// TIA Portal V15.1 export
// export: Created 2026-01-09T13:45:15.6924077Z, ExportSetting WithDefaults, WithReadOnly, DisplayName Totally Integrated Automation Portal, DisplayVersion V15.1 Update 8, DisplayName TIA Portal Openness, DisplayVersion V15.1 Update 8, DisplayName STEP 7 Professional, DisplayVersion V15.1 Update 8, DisplayName WinCC Advanced, DisplayVersion V15.1 Update 8
FUNCTION "FCXL_CCD_AP1" : Void   // FC15, LAD
{ S7_Optimized_Access := 'TRUE' }
VERSION : 0.1
// stored: AutoNumber true, CodeModifiedDate 2026-01-04T14:27:05.6438339Z, CompileDate 2026-01-04T14:27:05.690726Z, CreationDate 2024-10-13T15:07:34.9617085Z, HandleErrorsWithinBlock false, InterfaceModifiedDate 2024-08-08T03:23:40.7447783Z, IsConsistent true, IsIECCheckEnabled false, IsKnowHowProtected false, IsWriteProtected false, LibraryConformanceStatus Error: The block contains calls of single instances. Warning: The object contains access to global data blocks. Warning: The block contains direct access to inputs, outputs, bit memories, indirect access to the registry or indirect access to external memory areas that are unknown at the time of compilation., ModifiedDate 2026-01-04T14:27:05.6438339Z, ParameterModified 2024-08-08T03:23:40.7447783Z, PLCSimAdvancedSupport false, SetENOAutomatically False, StructureModified 2024-08-08T03:23:40.7447783Z, UDAEnableTagReadback false
   VAR_TEMP   // added for the SCL form of the ladder/FBD networks
      _w1 : Bool;
      _w2 : Bool;
      _w3 : Bool;
   END_VAR
BEGIN

REGION Network 1
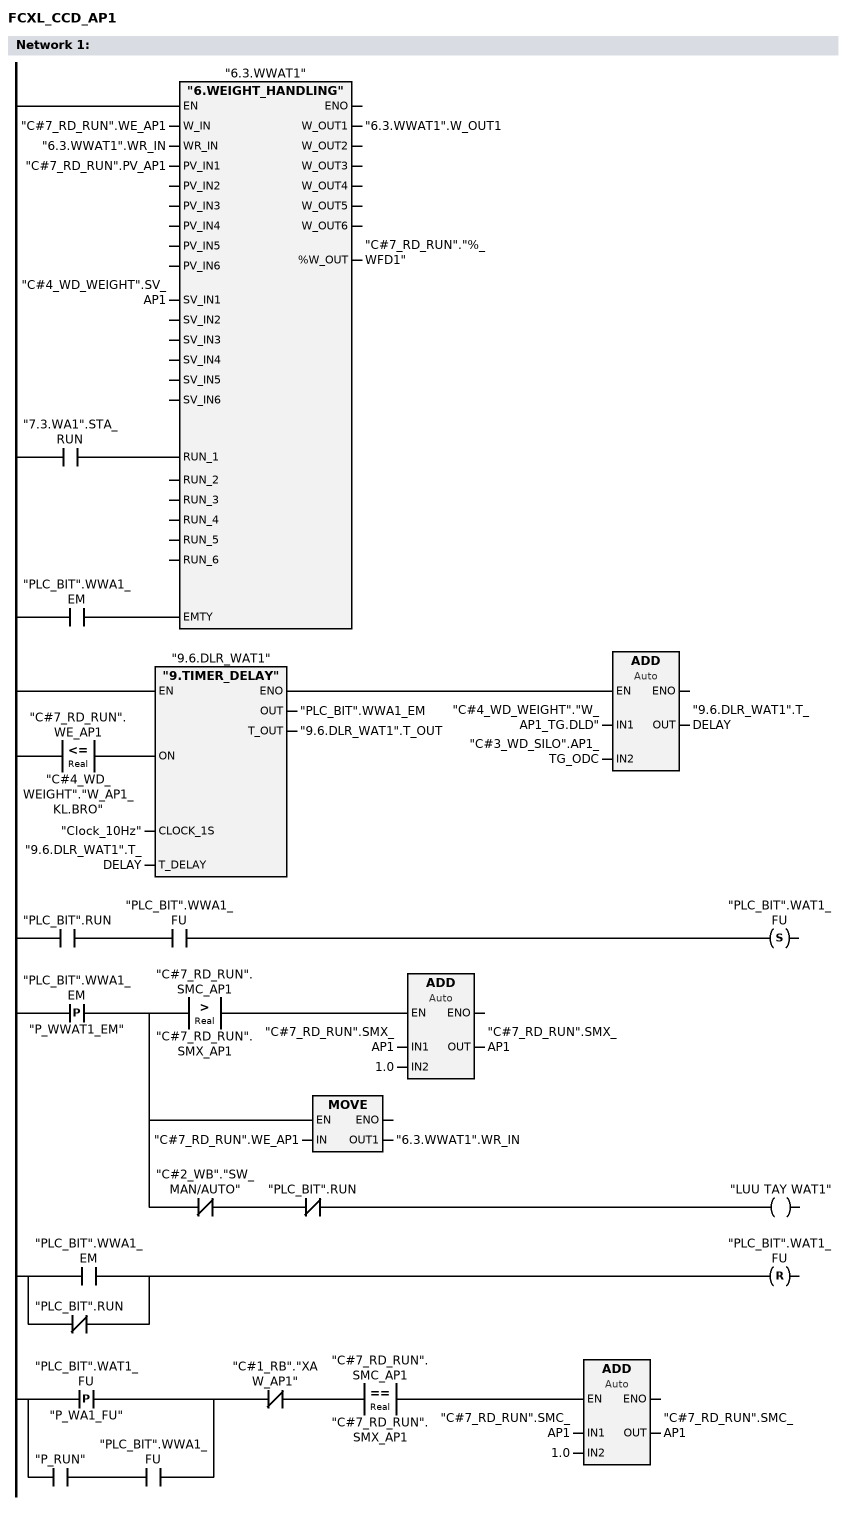
   RUNG wire#powerrail
      "6.3.WWAT1"(RUN_1 := wire#w1, EMTY := wire#w2, W_IN := "C#7_RD_RUN".WE_AP1, WR_IN := "6.3.WWAT1".WR_IN, PV_IN1 := "C#7_RD_RUN".PV_AP1, PV_IN2 :=, PV_IN3 :=, PV_IN4 :=, PV_IN5 :=, PV_IN6 :=, SV_IN1 := "C#4_WD_WEIGHT".SV_AP1, SV_IN2 :=, SV_IN3 :=, SV_IN4 :=, SV_IN5 :=, SV_IN6 :=, RUN_2 :=, RUN_3 :=, RUN_4 :=, RUN_5 :=, RUN_6 :=, W_OUT1 => "6.3.WWAT1".W_OUT1, W_OUT2 =>, W_OUT3 =>, W_OUT4 =>, W_OUT5 =>, W_OUT6 =>, "%W_OUT" => "C#7_RD_RUN"."%_WFD1")
   END_RUNG
   RUNG wire#powerrail
      Contact( "7.3.WA1".STA_RUN )
   END_RUNG wire#w1
   RUNG wire#powerrail
      Contact( "PLC_BIT".WWA1_EM )
   END_RUNG wire#w2
   RUNG wire#powerrail
      "9.6.DLR_WAT1"(ON := wire#w3, CLOCK_1S := "Clock_10Hz", T_DELAY := "9.6.DLR_WAT1".T_DELAY, OUT => "PLC_BIT".WWA1_EM, T_OUT => "9.6.DLR_WAT1".T_OUT)
      Add(in1 := "C#4_WD_WEIGHT"."W_AP1_TG.DLD", in2 := "C#3_WD_SILO".AP1_TG_ODC, out => "9.6.DLR_WAT1".T_DELAY)
   END_RUNG
   RUNG wire#powerrail
      { S7_Templates := "SrcType := Real" } LE_Contact(in1 := "C#7_RD_RUN".WE_AP1, in2 := "C#4_WD_WEIGHT"."W_AP1_KL.BRO")
   END_RUNG wire#w3
   RUNG wire#powerrail
      Contact( "PLC_BIT".RUN )
      Contact( "PLC_BIT".WWA1_FU )
      S_Coil( "PLC_BIT".WAT1_FU )
   END_RUNG
   RUNG wire#powerrail
      P_Contact(operand := "PLC_BIT".WWA1_EM, bit := "P_WWAT1_EM")
      wire#w4
      { S7_Templates := "SrcType := Real" } GT_Contact(in1 := "C#7_RD_RUN".SMC_AP1, in2 := "C#7_RD_RUN".SMX_AP1)
      Add(in1 := "C#7_RD_RUN".SMX_AP1, in2 := 1.0, out => "C#7_RD_RUN".SMX_AP1)
   END_RUNG
   RUNG wire#w4
      Move(in := "C#7_RD_RUN".WE_AP1, out1 => "6.3.WWAT1".WR_IN)
   END_RUNG
   RUNG wire#w4
      I_Contact( "C#2_WB"."SW_MAN/AUTO" )
      I_Contact( "PLC_BIT".RUN )
      Coil( "LUU TAY WAT1" )
   END_RUNG
   RUNG wire#powerrail
      Contact( "PLC_BIT".WWA1_EM )
      wire#w5
      R_Coil( "PLC_BIT".WAT1_FU )
   END_RUNG
   RUNG wire#powerrail
      I_Contact( "PLC_BIT".RUN )
   END_RUNG wire#w5
   RUNG wire#powerrail
      P_Contact(operand := "PLC_BIT".WAT1_FU, bit := "P_WA1_FU")
      wire#w6
      I_Contact( "C#1_RB"."XA W_AP1" )
      { S7_Templates := "SrcType := Real" } EQ_Contact(in1 := "C#7_RD_RUN".SMC_AP1, in2 := "C#7_RD_RUN".SMX_AP1)
      Add(in1 := "C#7_RD_RUN".SMC_AP1, in2 := 1.0, out => "C#7_RD_RUN".SMC_AP1)
   END_RUNG
   RUNG wire#powerrail
      Contact( "P_RUN" )
      Contact( "PLC_BIT".WWA1_FU )
   END_RUNG wire#w6
   // the same network as SCL:
   "6.3.WWAT1"(W_IN := "C#7_RD_RUN".WE_AP1,   // "6.WEIGHT_HANDLING"
               WR_IN := "6.3.WWAT1".WR_IN,
               PV_IN1 := "C#7_RD_RUN".PV_AP1,
               SV_IN1 := "C#4_WD_WEIGHT".SV_AP1,
               RUN_1 := "7.3.WA1".STA_RUN,
               EMTY := "PLC_BIT".WWA1_EM,
               W_OUT1 => "6.3.WWAT1".W_OUT1,
               "%W_OUT" => "C#7_RD_RUN"."%_WFD1");
   "9.6.DLR_WAT1"(ON := "C#7_RD_RUN".WE_AP1 <= "C#4_WD_WEIGHT"."W_AP1_KL.BRO",   // "9.TIMER_DELAY"
                  CLOCK_1S := "Clock_10Hz",
                  T_DELAY := "9.6.DLR_WAT1".T_DELAY,
                  OUT => "PLC_BIT".WWA1_EM,
                  T_OUT => "9.6.DLR_WAT1".T_OUT,
                  ENO => #_w1);
   IF #_w1 THEN "9.6.DLR_WAT1".T_DELAY := "C#4_WD_WEIGHT"."W_AP1_TG.DLD" + "C#3_WD_SILO".AP1_TG_ODC; END_IF;
   IF "PLC_BIT".RUN AND "PLC_BIT".WWA1_FU THEN "PLC_BIT".WAT1_FU := TRUE; END_IF;
   #_w2 := "PLC_BIT".WWA1_EM AND NOT "P_WWAT1_EM";   // rising edge of "PLC_BIT".WWA1_EM
   "P_WWAT1_EM" := "PLC_BIT".WWA1_EM;
   IF #_w2 AND ("C#7_RD_RUN".SMC_AP1 > "C#7_RD_RUN".SMX_AP1) THEN
       "C#7_RD_RUN".SMX_AP1 := "C#7_RD_RUN".SMX_AP1 + 1.0;
   END_IF;
   IF #_w2 THEN "6.3.WWAT1".WR_IN := "C#7_RD_RUN".WE_AP1; END_IF;
   "LUU TAY WAT1" := #_w2 AND NOT "C#2_WB"."SW_MAN/AUTO" AND NOT "PLC_BIT".RUN;
   IF "PLC_BIT".WWA1_EM OR NOT "PLC_BIT".RUN THEN "PLC_BIT".WAT1_FU := FALSE; END_IF;
   #_w3 := "PLC_BIT".WAT1_FU AND NOT "P_WA1_FU";   // rising edge of "PLC_BIT".WAT1_FU
   "P_WA1_FU" := "PLC_BIT".WAT1_FU;
   IF (#_w3 OR ("P_RUN" AND "PLC_BIT".WWA1_FU)) AND NOT "C#1_RB"."XA W_AP1" AND ("C#7_RD_RUN".SMC_AP1 = "C#7_RD_RUN".SMX_AP1) THEN
       "C#7_RD_RUN".SMC_AP1 := "C#7_RD_RUN".SMC_AP1 + 1.0;
   END_IF;
END_REGION
END_FUNCTION
